PROGRAM MAIN

VAR
	high : REAL;
	temp : REAL;
	conc : REAL;
END_VAR

// Make the calculations based on consistent data
high := NextHigh();
temp := NextTemp();
conc := NextConc();

// Update the globals
GVL.high_now := high;
GVL.temp_now := temp;
GVL.conc_now := conc;

// Update the CIP status
SetCIP(FALSE);

// Calculate time
GVL.time_now := RunTime();

GVL.alarm := CheckAlarm();


// HOW DOES THE TANK WALL WORK //

END_PROGRAM

(* stored: Version 1.1.0.1, ProductVersion 3.1.4024.12
   POU MAIN: Id {da1e2e68-f202-4ed0-8d51-9abdfc0ccaa5}, SpecialFunc None *)
